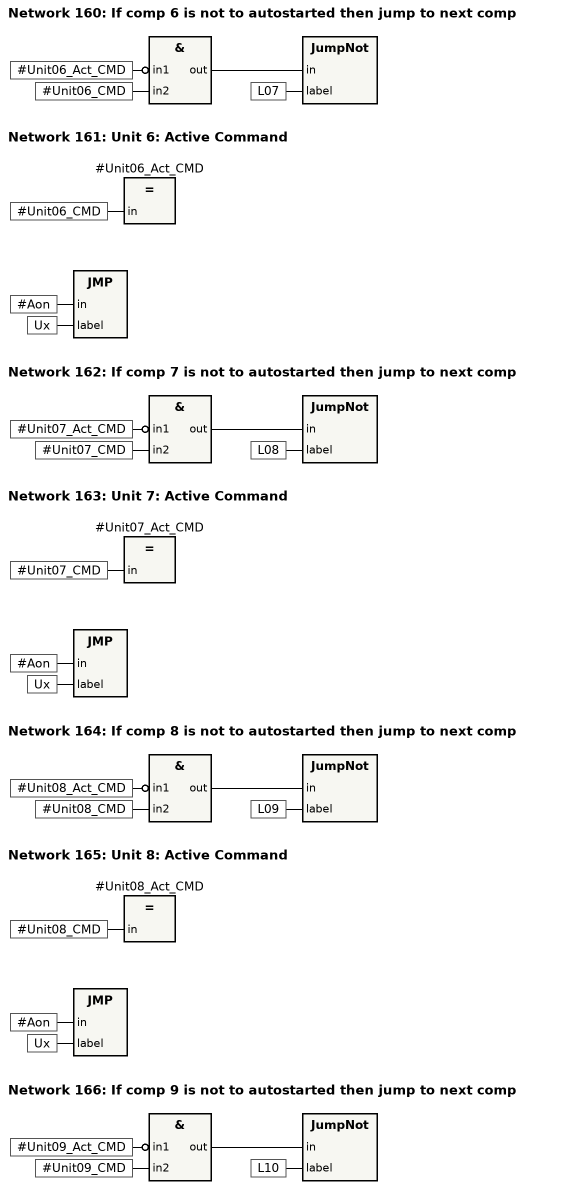
   // no SCL statement known for JumpNot: written as a call
   L06:
   JumpNot(in := NOT #Unit06_Act_CMD AND #Unit06_CMD, label := L07);
END_REGION

REGION Network 161: Unit 6: Active Command
   // Jump to end
   #Unit06_Act_CMD := #Unit06_CMD;
   IF #Aon THEN GOTO Ux; END_IF;
END_REGION

REGION Network 162: If comp 7 is not to autostarted then jump to next comp
   // no SCL statement known for JumpNot: written as a call
   L07:
   JumpNot(in := NOT #Unit07_Act_CMD AND #Unit07_CMD, label := L08);
END_REGION

REGION Network 163: Unit 7: Active Command
   // Jump to end
   #Unit07_Act_CMD := #Unit07_CMD;
   IF #Aon THEN GOTO Ux; END_IF;
END_REGION

REGION Network 164: If comp 8 is not to autostarted then jump to next comp
   // no SCL statement known for JumpNot: written as a call
   L08:
   JumpNot(in := NOT #Unit08_Act_CMD AND #Unit08_CMD, label := L09);
END_REGION

REGION Network 165: Unit 8: Active Command
   // Jump to end
   #Unit08_Act_CMD := #Unit08_CMD;
   IF #Aon THEN GOTO Ux; END_IF;
END_REGION

REGION Network 166: If comp 9 is not to autostarted then jump to next comp
   // no SCL statement known for JumpNot: written as a call
   L09:
   JumpNot(in := NOT #Unit09_Act_CMD AND #Unit09_CMD, label := L10);
END_REGION

REGION Network 167: Unit 9: Active Command
   // Jump to end
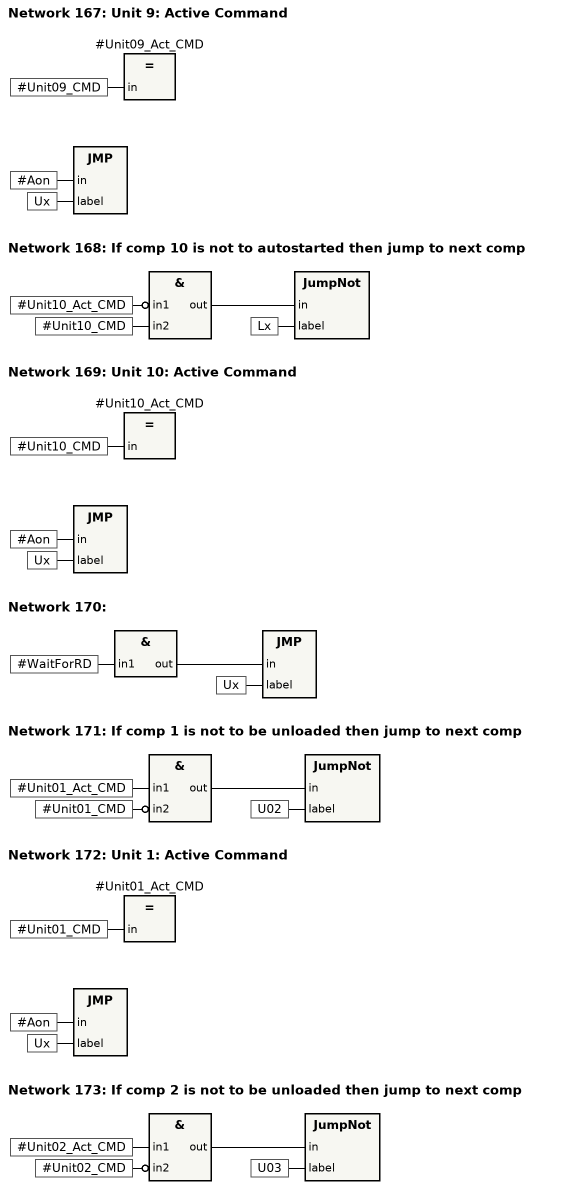
   #Unit09_Act_CMD := #Unit09_CMD;
   IF #Aon THEN GOTO Ux; END_IF;
END_REGION

REGION Network 168: If comp 10 is not to autostarted then jump to next comp
   // no SCL statement known for JumpNot: written as a call
   L10:
   JumpNot(in := NOT #Unit10_Act_CMD AND #Unit10_CMD, label := Lx);
END_REGION

REGION Network 169: Unit 10: Active Command
   // Jump to end
   #Unit10_Act_CMD := #Unit10_CMD;
   IF #Aon THEN GOTO Ux; END_IF;
END_REGION

REGION Network 170
   Lx:
   IF #WaitForRD THEN GOTO Ux; END_IF;
END_REGION

REGION Network 171: If comp 1 is not to be unloaded then jump to next comp
   // no SCL statement known for JumpNot: written as a call
   JumpNot(in := #Unit01_Act_CMD AND NOT #Unit01_CMD, label := U02);
END_REGION

REGION Network 172: Unit 1: Active Command
   #Unit01_Act_CMD := #Unit01_CMD;
   IF #Aon THEN GOTO Ux; END_IF;
END_REGION

REGION Network 173: If comp 2 is not to be unloaded then jump to next comp
   // no SCL statement known for JumpNot: written as a call
   U02:
   JumpNot(in := #Unit02_Act_CMD AND NOT #Unit02_CMD, label := U03);
END_REGION

REGION Network 174: Unit 2: Active Command
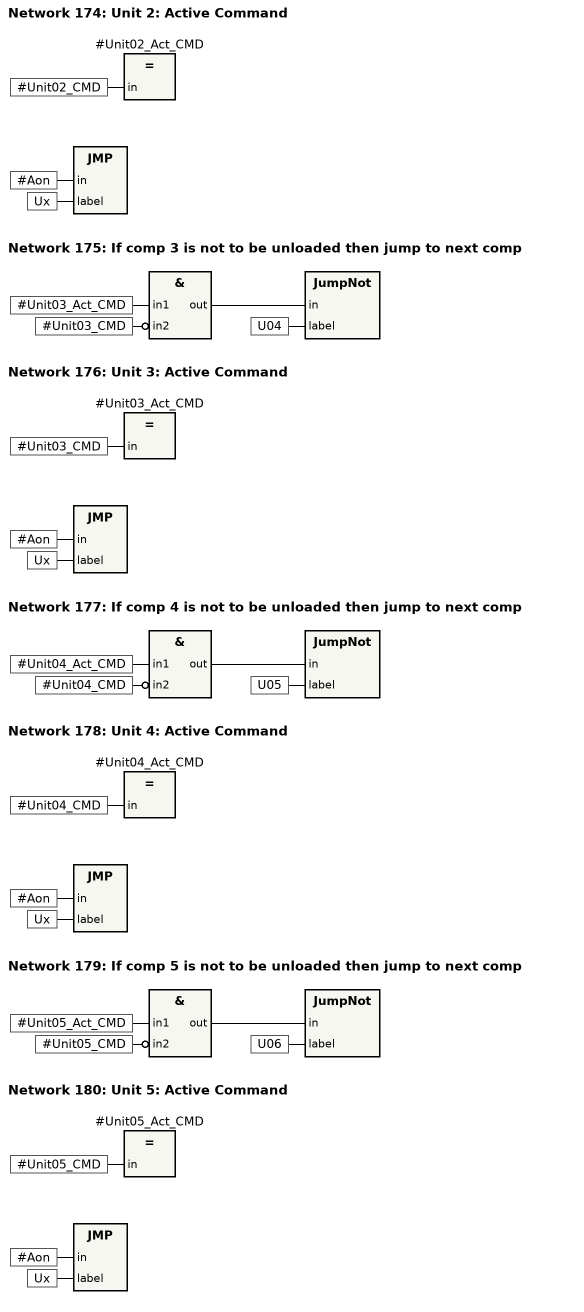
   #Unit02_Act_CMD := #Unit02_CMD;
   IF #Aon THEN GOTO Ux; END_IF;
END_REGION

REGION Network 175: If comp 3 is not to be unloaded then jump to next comp
   // no SCL statement known for JumpNot: written as a call
   U03:
   JumpNot(in := #Unit03_Act_CMD AND NOT #Unit03_CMD, label := U04);
END_REGION

REGION Network 176: Unit 3: Active Command
   #Unit03_Act_CMD := #Unit03_CMD;
   IF #Aon THEN GOTO Ux; END_IF;
END_REGION

REGION Network 177: If comp 4 is not to be unloaded then jump to next comp
   // no SCL statement known for JumpNot: written as a call
   U04:
   JumpNot(in := #Unit04_Act_CMD AND NOT #Unit04_CMD, label := U05);
END_REGION

REGION Network 178: Unit 4: Active Command
   #Unit04_Act_CMD := #Unit04_CMD;
   IF #Aon THEN GOTO Ux; END_IF;
END_REGION

REGION Network 179: If comp 5 is not to be unloaded then jump to next comp
   // no SCL statement known for JumpNot: written as a call
   U05:
   JumpNot(in := #Unit05_Act_CMD AND NOT #Unit05_CMD, label := U06);
END_REGION

REGION Network 180: Unit 5: Active Command
   #Unit05_Act_CMD := #Unit05_CMD;
   IF #Aon THEN GOTO Ux; END_IF;
END_REGION

REGION Network 181: If comp 6 is not to be unloaded then jump to next comp
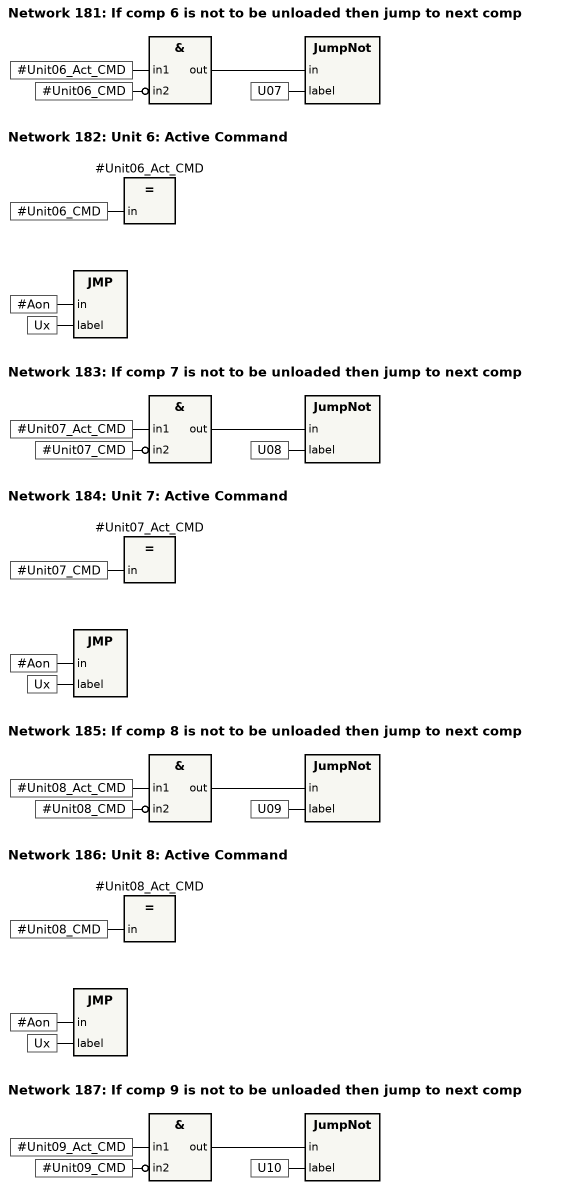
   // no SCL statement known for JumpNot: written as a call
   U06:
   JumpNot(in := #Unit06_Act_CMD AND NOT #Unit06_CMD, label := U07);
END_REGION

REGION Network 182: Unit 6: Active Command
   #Unit06_Act_CMD := #Unit06_CMD;
   IF #Aon THEN GOTO Ux; END_IF;
END_REGION

REGION Network 183: If comp 7 is not to be unloaded then jump to next comp
   // no SCL statement known for JumpNot: written as a call
   U07:
   JumpNot(in := #Unit07_Act_CMD AND NOT #Unit07_CMD, label := U08);
END_REGION

REGION Network 184: Unit 7: Active Command
   #Unit07_Act_CMD := #Unit07_CMD;
   IF #Aon THEN GOTO Ux; END_IF;
END_REGION

REGION Network 185: If comp 8 is not to be unloaded then jump to next comp
   // no SCL statement known for JumpNot: written as a call
   U08:
   JumpNot(in := #Unit08_Act_CMD AND NOT #Unit08_CMD, label := U09);
END_REGION

REGION Network 186: Unit 8: Active Command
   #Unit08_Act_CMD := #Unit08_CMD;
   IF #Aon THEN GOTO Ux; END_IF;
END_REGION

REGION Network 187: If comp 9 is not to be unloaded then jump to next comp
   // no SCL statement known for JumpNot: written as a call
   U09:
   JumpNot(in := #Unit09_Act_CMD AND NOT #Unit09_CMD, label := U10);
END_REGION

REGION Network 188: Unit 9: Active Command
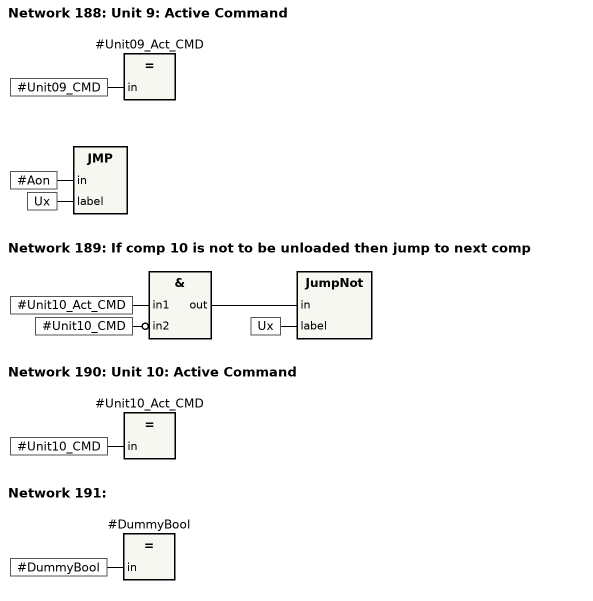
   #Unit09_Act_CMD := #Unit09_CMD;
   IF #Aon THEN GOTO Ux; END_IF;
END_REGION

REGION Network 189: If comp 10 is not to be unloaded then jump to next comp
   // no SCL statement known for JumpNot: written as a call
   U10:
   JumpNot(in := #Unit10_Act_CMD AND NOT #Unit10_CMD, label := Ux);
END_REGION

REGION Network 190: Unit 10: Active Command
   #Unit10_Act_CMD := #Unit10_CMD;
END_REGION

REGION Network 191
   Ux:
   #DummyBool := #DummyBool;
END_REGION

REGION Network 192: Reset Active commands if not selected, SACK or OK
   // Every x s a compressor is unloaded and one is loaded
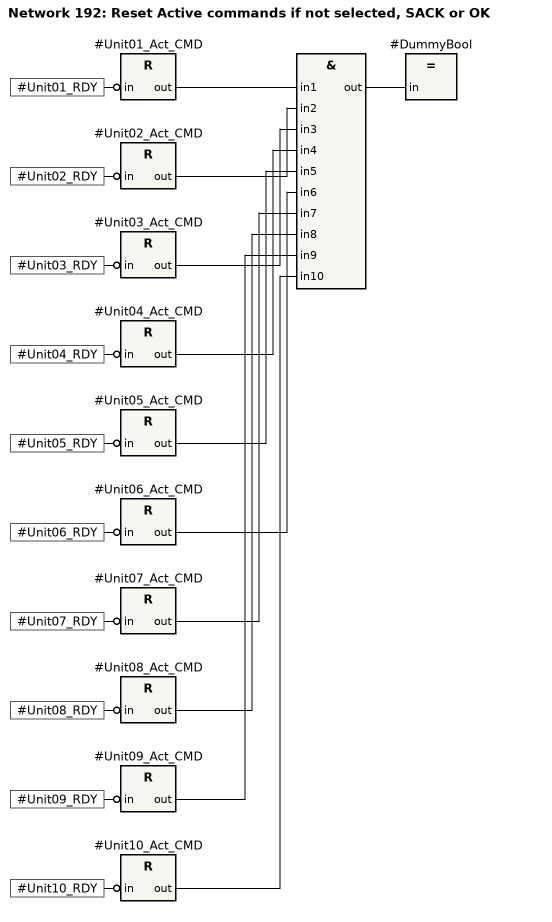
   IF NOT #Unit01_RDY THEN #Unit01_Act_CMD := FALSE; END_IF;
   IF NOT #Unit02_RDY THEN #Unit02_Act_CMD := FALSE; END_IF;
   IF NOT #Unit03_RDY THEN #Unit03_Act_CMD := FALSE; END_IF;
   IF NOT #Unit04_RDY THEN #Unit04_Act_CMD := FALSE; END_IF;
   IF NOT #Unit05_RDY THEN #Unit05_Act_CMD := FALSE; END_IF;
   IF NOT #Unit06_RDY THEN #Unit06_Act_CMD := FALSE; END_IF;
   IF NOT #Unit07_RDY THEN #Unit07_Act_CMD := FALSE; END_IF;
   IF NOT #Unit08_RDY THEN #Unit08_Act_CMD := FALSE; END_IF;
   IF NOT #Unit09_RDY THEN #Unit09_Act_CMD := FALSE; END_IF;
   IF NOT #Unit10_RDY THEN #Unit10_Act_CMD := FALSE; END_IF;
   #DummyBool := NOT #Unit01_RDY AND NOT #Unit02_RDY AND NOT #Unit03_RDY AND NOT #Unit04_RDY AND NOT #Unit05_RDY AND NOT #Unit06_RDY AND NOT #Unit07_RDY AND NOT #Unit08_RDY AND NOT #Unit09_RDY AND NOT #Unit10_RDY;
END_REGION

REGION Network 193: 12) Set Load Commands
   // Build 002 - 28 June.2019 (EXTBOB): Load outputs can only be energized if selected from faceplate
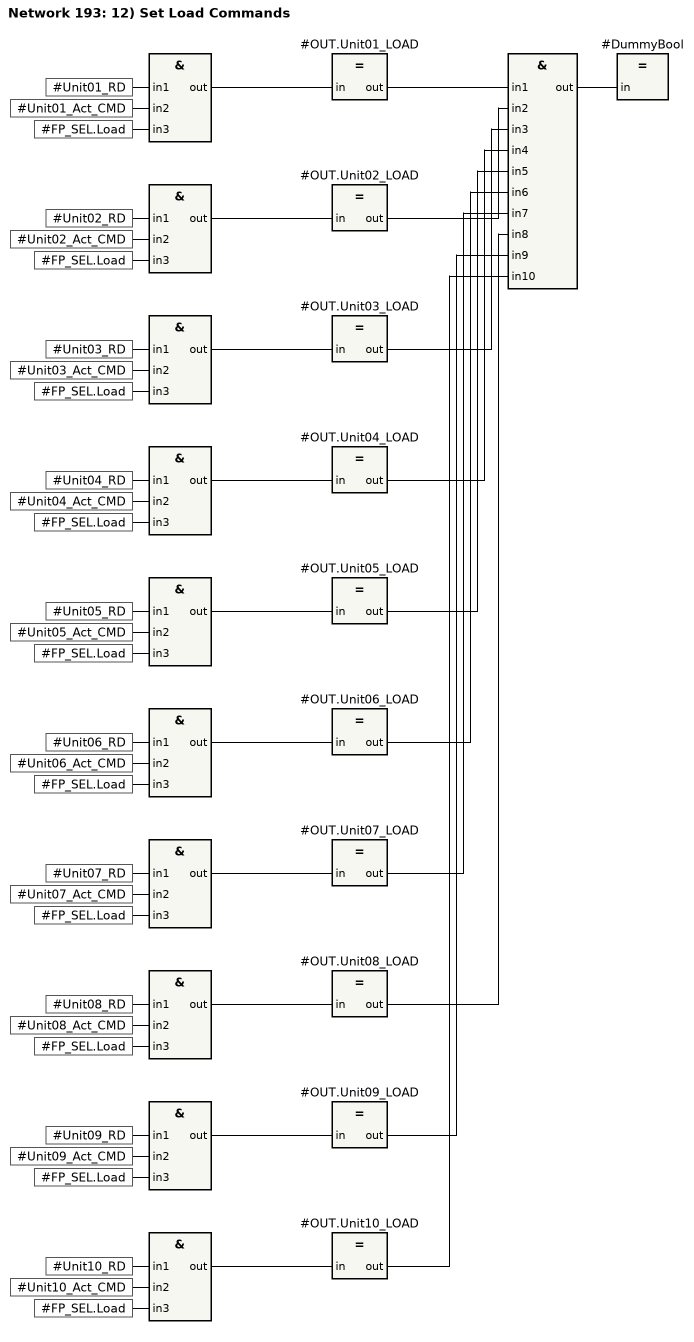
   #OUT.Unit01_LOAD := #Unit01_RD AND #Unit01_Act_CMD AND #FP_SEL.Load;
   #OUT.Unit02_LOAD := #Unit02_RD AND #Unit02_Act_CMD AND #FP_SEL.Load;
   #OUT.Unit03_LOAD := #Unit03_RD AND #Unit03_Act_CMD AND #FP_SEL.Load;
   #OUT.Unit04_LOAD := #Unit04_RD AND #Unit04_Act_CMD AND #FP_SEL.Load;
   #OUT.Unit05_LOAD := #Unit05_RD AND #Unit05_Act_CMD AND #FP_SEL.Load;
   #OUT.Unit06_LOAD := #Unit06_RD AND #Unit06_Act_CMD AND #FP_SEL.Load;
   #OUT.Unit07_LOAD := #Unit07_RD AND #Unit07_Act_CMD AND #FP_SEL.Load;
   #OUT.Unit08_LOAD := #Unit08_RD AND #Unit08_Act_CMD AND #FP_SEL.Load;
   #OUT.Unit09_LOAD := #Unit09_RD AND #Unit09_Act_CMD AND #FP_SEL.Load;
   #OUT.Unit10_LOAD := #Unit10_RD AND #Unit10_Act_CMD AND #FP_SEL.Load;
   #DummyBool := #OUT.Unit01_LOAD AND #OUT.Unit02_LOAD AND #OUT.Unit03_LOAD AND #OUT.Unit04_LOAD AND #OUT.Unit05_LOAD AND #OUT.Unit06_LOAD AND #OUT.Unit07_LOAD AND #OUT.Unit08_LOAD AND #OUT.Unit09_LOAD AND #OUT.Unit10_LOAD;
END_REGION

REGION Network 194: Set ASTR Output (Delayed off)
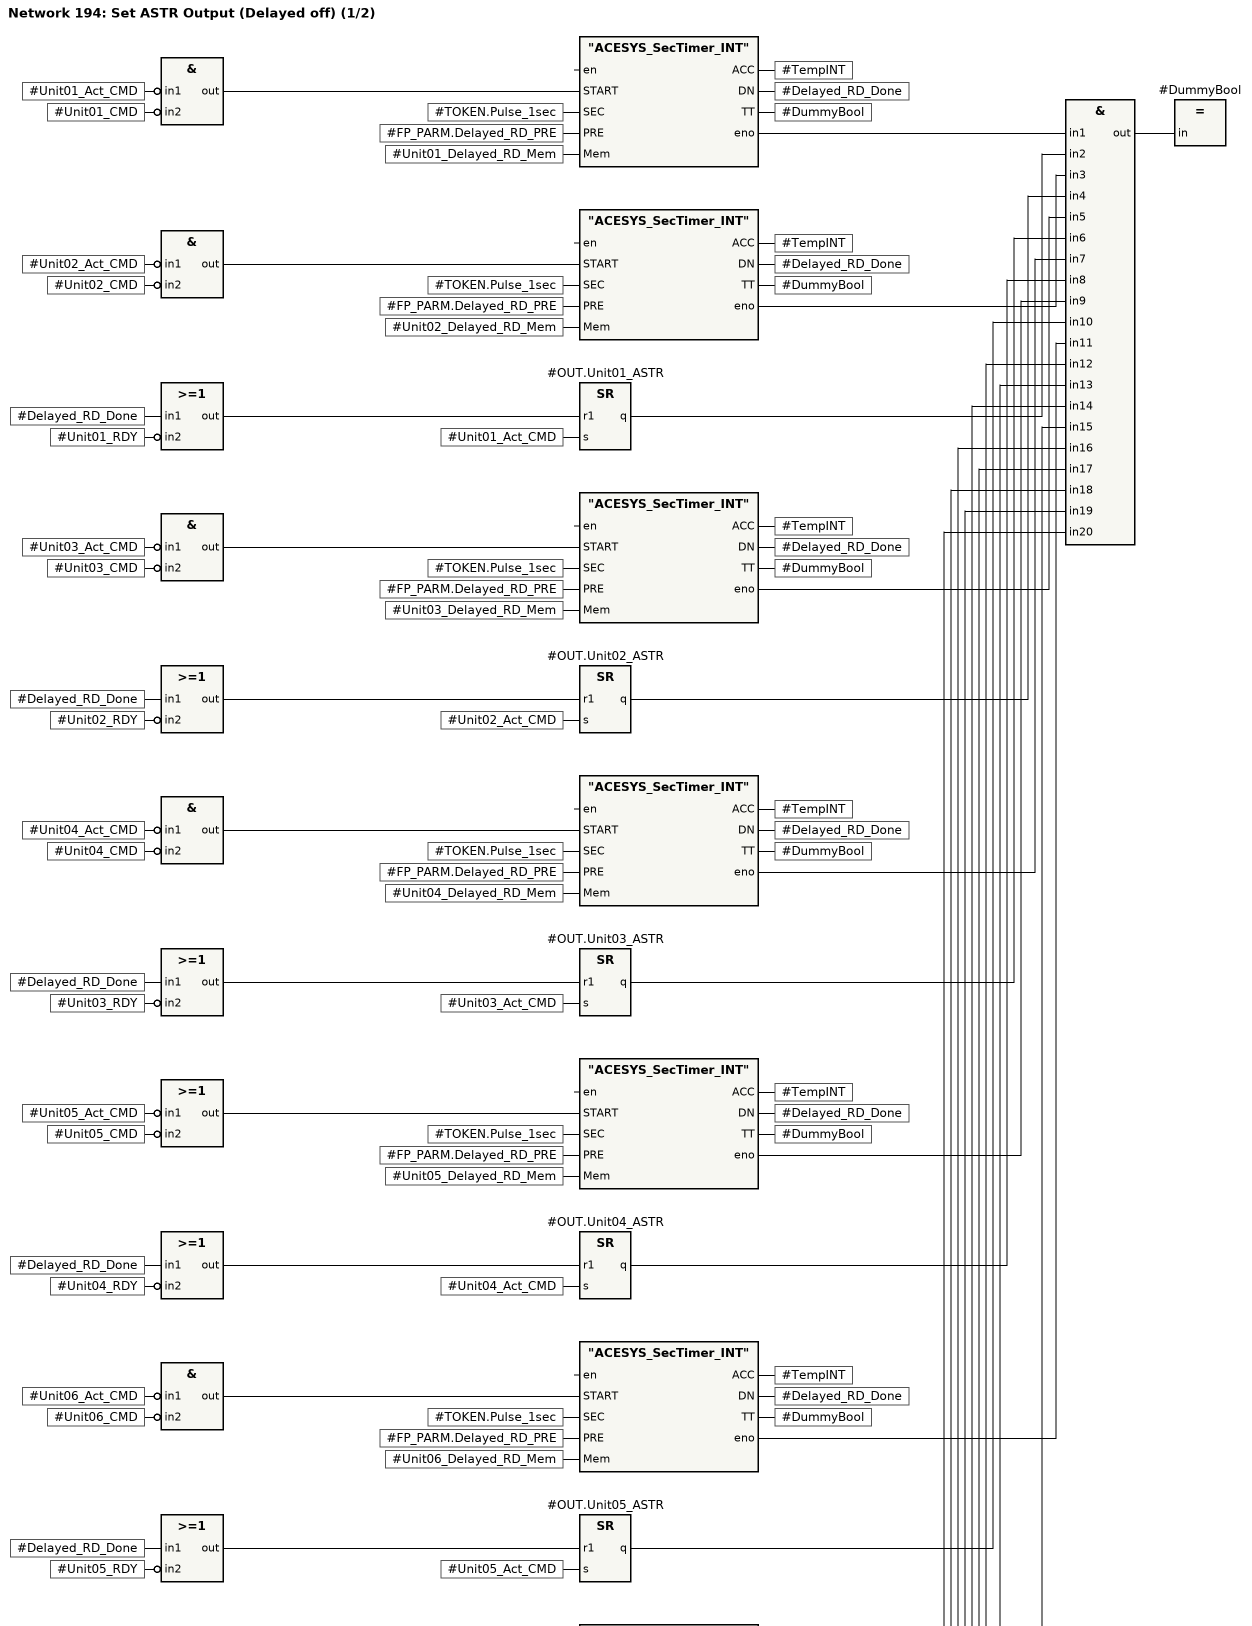
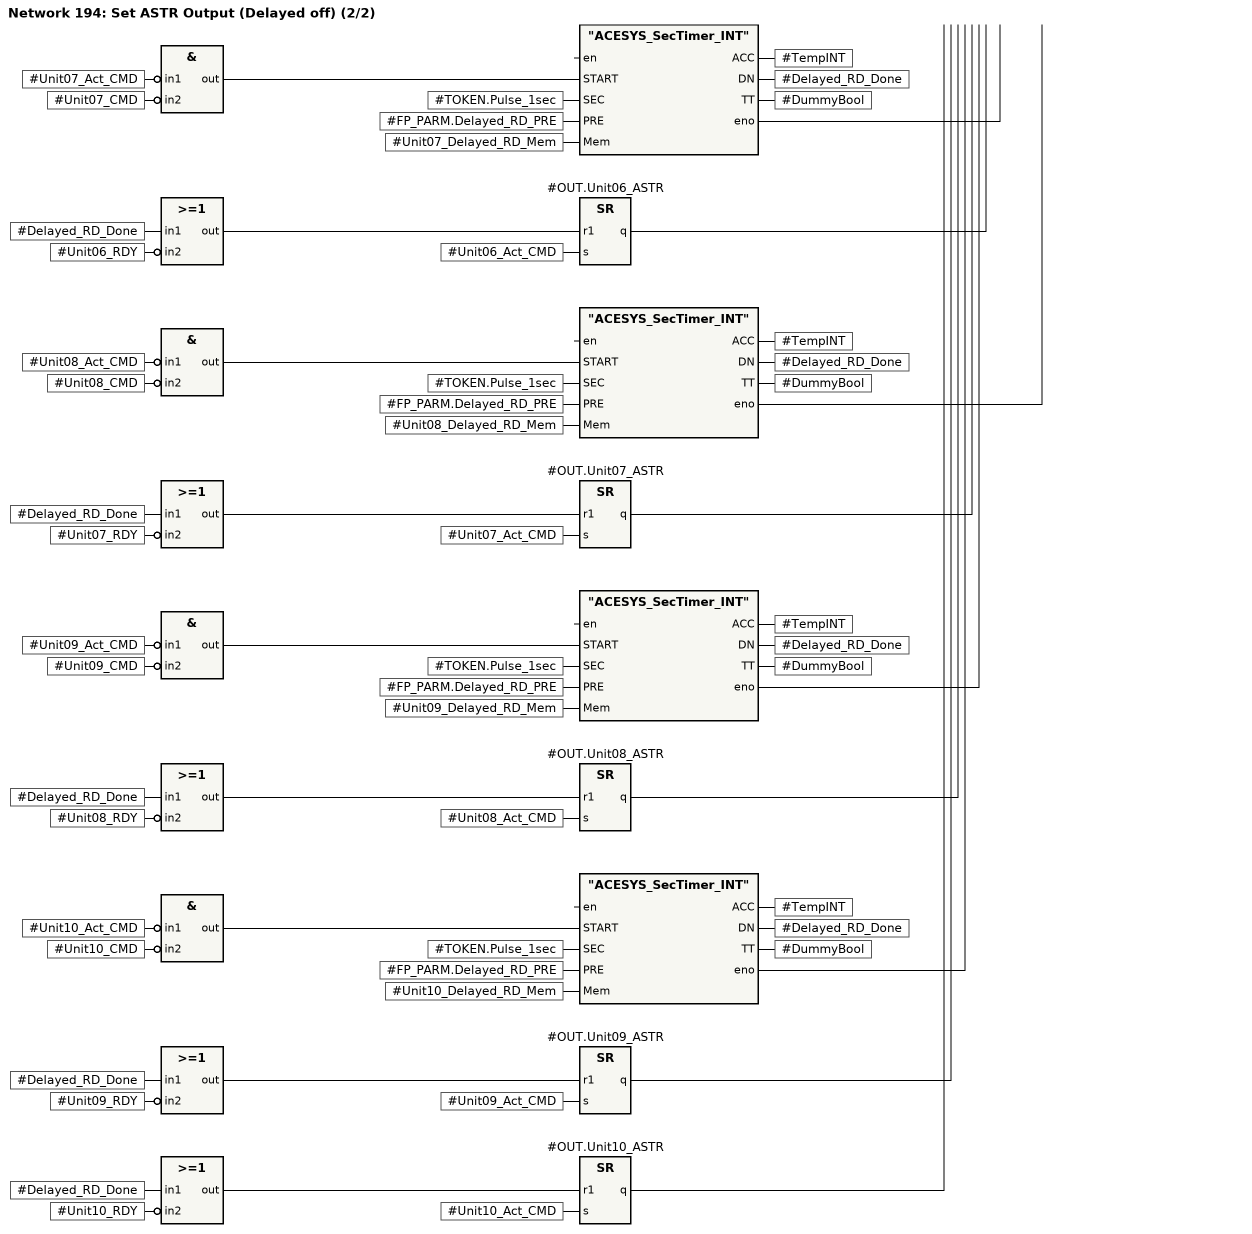
   "ACESYS_SecTimer_INT"(START := NOT #Unit01_Act_CMD AND NOT #Unit01_CMD,
                         SEC := #TOKEN.Pulse_1sec,
                         PRE := #FP_PARM.Delayed_RD_PRE,
                         Mem := #Unit01_Delayed_RD_Mem,
                         ACC => #TempINT,
                         DN => #Delayed_RD_Done,
                         TT => #DummyBool,
                         ENO => #_w1);
   IF #Unit01_Act_CMD THEN
       #OUT.Unit01_ASTR := TRUE;   // SR flip-flop
   END_IF;
   IF #Delayed_RD_Done OR NOT #Unit01_RDY THEN #OUT.Unit01_ASTR := FALSE; END_IF;
   "ACESYS_SecTimer_INT"(START := NOT #Unit02_Act_CMD AND NOT #Unit02_CMD,
                         SEC := #TOKEN.Pulse_1sec,
                         PRE := #FP_PARM.Delayed_RD_PRE,
                         Mem := #Unit02_Delayed_RD_Mem,
                         ACC => #TempINT,
                         DN => #Delayed_RD_Done,
                         TT => #DummyBool,
                         ENO => #_w2);
   IF #Unit02_Act_CMD THEN
       #OUT.Unit02_ASTR := TRUE;   // SR flip-flop
   END_IF;
   IF #Delayed_RD_Done OR NOT #Unit02_RDY THEN #OUT.Unit02_ASTR := FALSE; END_IF;
   "ACESYS_SecTimer_INT"(START := NOT #Unit03_Act_CMD AND NOT #Unit03_CMD,
                         SEC := #TOKEN.Pulse_1sec,
                         PRE := #FP_PARM.Delayed_RD_PRE,
                         Mem := #Unit03_Delayed_RD_Mem,
                         ACC => #TempINT,
                         DN => #Delayed_RD_Done,
                         TT => #DummyBool,
                         ENO => #_w3);
   IF #Unit03_Act_CMD THEN
       #OUT.Unit03_ASTR := TRUE;   // SR flip-flop
   END_IF;
   IF #Delayed_RD_Done OR NOT #Unit03_RDY THEN #OUT.Unit03_ASTR := FALSE; END_IF;
   "ACESYS_SecTimer_INT"(START := NOT #Unit04_Act_CMD AND NOT #Unit04_CMD,
                         SEC := #TOKEN.Pulse_1sec,
                         PRE := #FP_PARM.Delayed_RD_PRE,
                         Mem := #Unit04_Delayed_RD_Mem,
                         ACC => #TempINT,
                         DN => #Delayed_RD_Done,
                         TT => #DummyBool,
                         ENO => #_w4);
   IF #Unit04_Act_CMD THEN
       #OUT.Unit04_ASTR := TRUE;   // SR flip-flop
   END_IF;
   IF #Delayed_RD_Done OR NOT #Unit04_RDY THEN #OUT.Unit04_ASTR := FALSE; END_IF;
   "ACESYS_SecTimer_INT"(START := NOT #Unit05_Act_CMD OR NOT #Unit05_CMD,
                         SEC := #TOKEN.Pulse_1sec,
                         PRE := #FP_PARM.Delayed_RD_PRE,
                         Mem := #Unit05_Delayed_RD_Mem,
                         ACC => #TempINT,
                         DN => #Delayed_RD_Done,
                         TT => #DummyBool,
                         ENO => #_w5);
   IF #Unit05_Act_CMD THEN
       #OUT.Unit05_ASTR := TRUE;   // SR flip-flop
   END_IF;
   IF #Delayed_RD_Done OR NOT #Unit05_RDY THEN #OUT.Unit05_ASTR := FALSE; END_IF;
   "ACESYS_SecTimer_INT"(START := NOT #Unit06_Act_CMD AND NOT #Unit06_CMD,
                         SEC := #TOKEN.Pulse_1sec,
                         PRE := #FP_PARM.Delayed_RD_PRE,
                         Mem := #Unit06_Delayed_RD_Mem,
                         ACC => #TempINT,
                         DN => #Delayed_RD_Done,
                         TT => #DummyBool,
                         ENO => #_w6);
   IF #Unit06_Act_CMD THEN
       #OUT.Unit06_ASTR := TRUE;   // SR flip-flop
   END_IF;
   IF #Delayed_RD_Done OR NOT #Unit06_RDY THEN #OUT.Unit06_ASTR := FALSE; END_IF;
   "ACESYS_SecTimer_INT"(START := NOT #Unit07_Act_CMD AND NOT #Unit07_CMD,
                         SEC := #TOKEN.Pulse_1sec,
                         PRE := #FP_PARM.Delayed_RD_PRE,
                         Mem := #Unit07_Delayed_RD_Mem,
                         ACC => #TempINT,
                         DN => #Delayed_RD_Done,
                         TT => #DummyBool,
                         ENO => #_w7);
   IF #Unit07_Act_CMD THEN
       #OUT.Unit07_ASTR := TRUE;   // SR flip-flop
   END_IF;
   IF #Delayed_RD_Done OR NOT #Unit07_RDY THEN #OUT.Unit07_ASTR := FALSE; END_IF;
   "ACESYS_SecTimer_INT"(START := NOT #Unit08_Act_CMD AND NOT #Unit08_CMD,
                         SEC := #TOKEN.Pulse_1sec,
                         PRE := #FP_PARM.Delayed_RD_PRE,
                         Mem := #Unit08_Delayed_RD_Mem,
                         ACC => #TempINT,
                         DN => #Delayed_RD_Done,
                         TT => #DummyBool,
                         ENO => #_w8);
   IF #Unit08_Act_CMD THEN
       #OUT.Unit08_ASTR := TRUE;   // SR flip-flop
   END_IF;
   IF #Delayed_RD_Done OR NOT #Unit08_RDY THEN #OUT.Unit08_ASTR := FALSE; END_IF;
   "ACESYS_SecTimer_INT"(START := NOT #Unit09_Act_CMD AND NOT #Unit09_CMD,
                         SEC := #TOKEN.Pulse_1sec,
                         PRE := #FP_PARM.Delayed_RD_PRE,
                         Mem := #Unit09_Delayed_RD_Mem,
                         ACC => #TempINT,
                         DN => #Delayed_RD_Done,
                         TT => #DummyBool,
                         ENO => #_w9);
   IF #Unit09_Act_CMD THEN
       #OUT.Unit09_ASTR := TRUE;   // SR flip-flop
   END_IF;
   IF #Delayed_RD_Done OR NOT #Unit09_RDY THEN #OUT.Unit09_ASTR := FALSE; END_IF;
   "ACESYS_SecTimer_INT"(START := NOT #Unit10_Act_CMD AND NOT #Unit10_CMD,
                         SEC := #TOKEN.Pulse_1sec,
                         PRE := #FP_PARM.Delayed_RD_PRE,
                         Mem := #Unit10_Delayed_RD_Mem,
                         ACC => #TempINT,
                         DN => #Delayed_RD_Done,
                         TT => #DummyBool,
                         ENO => #_w10);
   IF #Unit10_Act_CMD THEN
       #OUT.Unit10_ASTR := TRUE;   // SR flip-flop
   END_IF;
   IF #Delayed_RD_Done OR NOT #Unit10_RDY THEN #OUT.Unit10_ASTR := FALSE; END_IF;
   #DummyBool := #_w1 AND #OUT.Unit01_ASTR AND #_w2 AND #OUT.Unit02_ASTR AND #_w3 AND #OUT.Unit03_ASTR AND #_w4 AND #OUT.Unit04_ASTR AND #_w5 AND #OUT.Unit05_ASTR AND #_w6 AND #OUT.Unit06_ASTR AND #_w7 AND #OUT.Unit07_ASTR AND #_w8 AND #OUT.Unit08_ASTR AND #_w9 AND #OUT.Unit09_ASTR AND #_w10 AND #OUT.Unit10_ASTR;
END_REGION

REGION Network 195
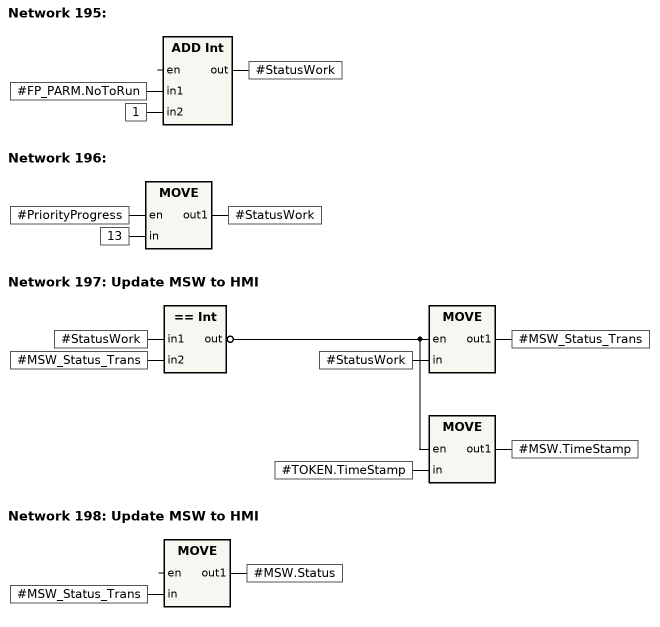
   #StatusWork := #FP_PARM.NoToRun + 1;
END_REGION

REGION Network 196
   IF #PriorityProgress THEN #StatusWork := 13; END_IF;
END_REGION

REGION Network 197: Update MSW to HMI
   #_w1 := NOT (#StatusWork = #MSW_Status_Trans);
   IF #_w1 THEN
       #MSW_Status_Trans := #StatusWork;
       #MSW.TimeStamp := #TOKEN.TimeStamp;
   END_IF;
END_REGION

REGION Network 198: Update MSW to HMI
   #MSW.Status := #MSW_Status_Trans;
END_REGION

REGION Network 199: Write STAT to OUT
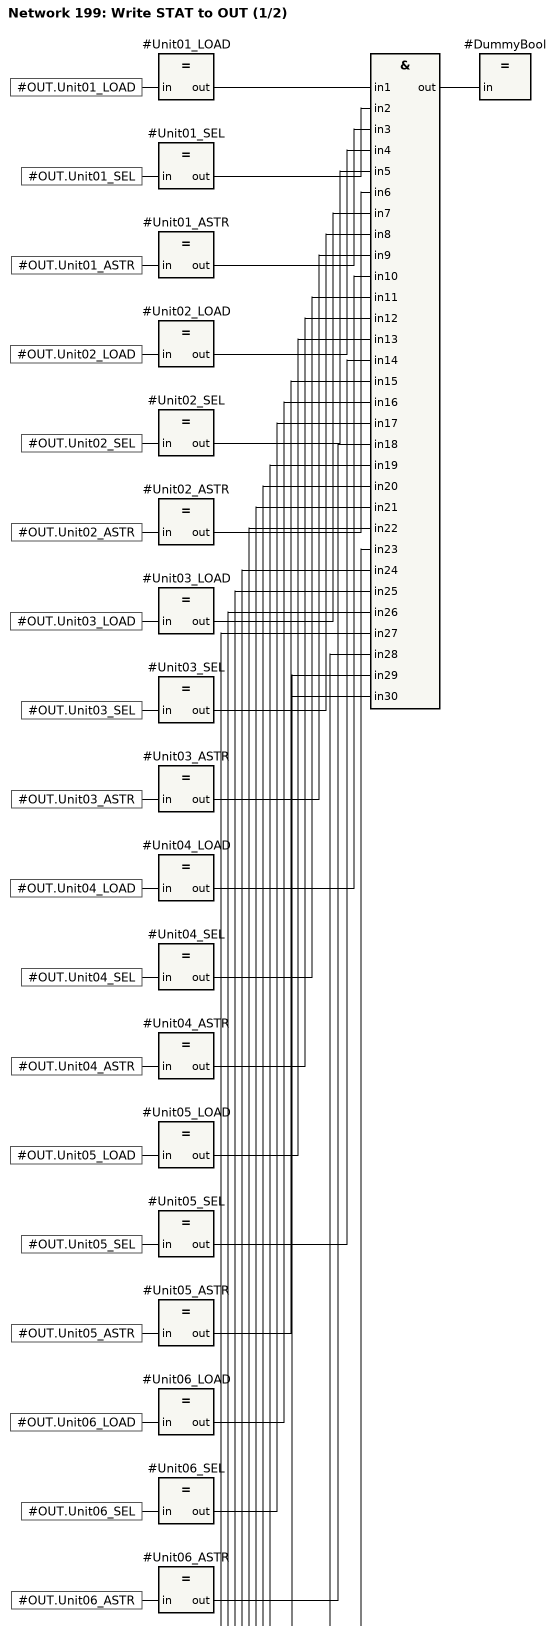
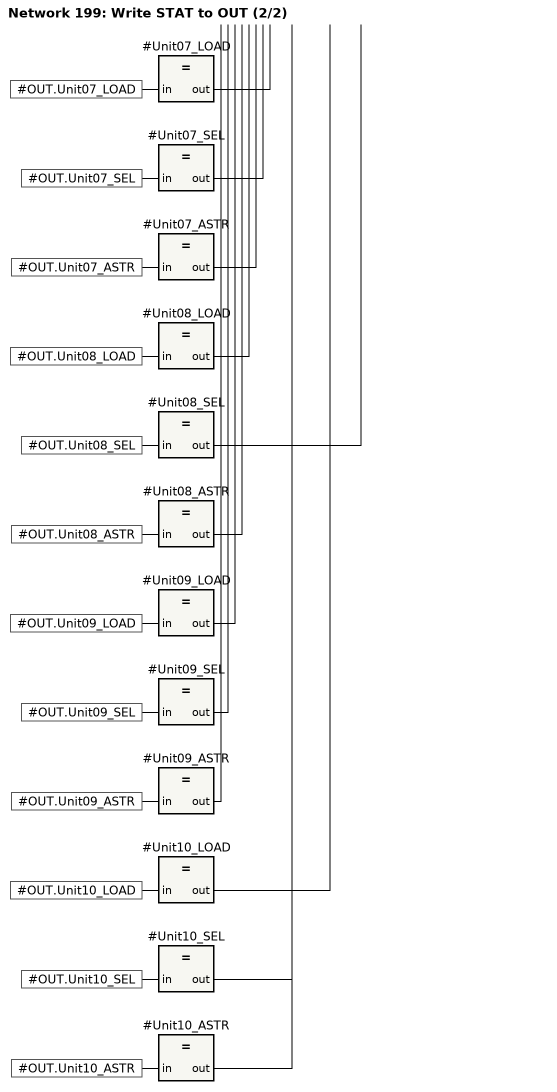
   #Unit01_LOAD := #OUT.Unit01_LOAD;
   #Unit01_SEL := #OUT.Unit01_SEL;
   #Unit01_ASTR := #OUT.Unit01_ASTR;
   #Unit02_LOAD := #OUT.Unit02_LOAD;
   #Unit02_SEL := #OUT.Unit02_SEL;
   #Unit02_ASTR := #OUT.Unit02_ASTR;
   #Unit03_LOAD := #OUT.Unit03_LOAD;
   #Unit03_SEL := #OUT.Unit03_SEL;
   #Unit03_ASTR := #OUT.Unit03_ASTR;
   #Unit04_LOAD := #OUT.Unit04_LOAD;
   #Unit04_SEL := #OUT.Unit04_SEL;
   #Unit04_ASTR := #OUT.Unit04_ASTR;
   #Unit05_LOAD := #OUT.Unit05_LOAD;
   #Unit05_SEL := #OUT.Unit05_SEL;
   #Unit05_ASTR := #OUT.Unit05_ASTR;
   #Unit06_LOAD := #OUT.Unit06_LOAD;
   #Unit06_SEL := #OUT.Unit06_SEL;
   #Unit06_ASTR := #OUT.Unit06_ASTR;
   #Unit07_LOAD := #OUT.Unit07_LOAD;
   #Unit07_SEL := #OUT.Unit07_SEL;
   #Unit07_ASTR := #OUT.Unit07_ASTR;
   #Unit08_LOAD := #OUT.Unit08_LOAD;
   #Unit08_SEL := #OUT.Unit08_SEL;
   #Unit08_ASTR := #OUT.Unit08_ASTR;
   #Unit09_LOAD := #OUT.Unit09_LOAD;
   #Unit09_SEL := #OUT.Unit09_SEL;
   #Unit09_ASTR := #OUT.Unit09_ASTR;
   #Unit10_LOAD := #OUT.Unit10_LOAD;
   #Unit10_SEL := #OUT.Unit10_SEL;
   #Unit10_ASTR := #OUT.Unit10_ASTR;
   #DummyBool := #OUT.Unit01_LOAD AND #OUT.Unit01_SEL AND #OUT.Unit01_ASTR AND #OUT.Unit02_LOAD AND #OUT.Unit02_SEL AND #OUT.Unit02_ASTR AND #OUT.Unit03_LOAD AND #OUT.Unit03_SEL AND #OUT.Unit03_ASTR AND #OUT.Unit04_LOAD AND #OUT.Unit04_SEL AND #OUT.Unit04_ASTR AND #OUT.Unit05_LOAD AND #OUT.Unit05_SEL AND #OUT.Unit05_ASTR AND #OUT.Unit06_LOAD AND #OUT.Unit06_SEL AND #OUT.Unit06_ASTR AND #OUT.Unit07_LOAD AND #OUT.Unit07_SEL AND #OUT.Unit07_ASTR AND #OUT.Unit08_LOAD AND #OUT.Unit08_SEL AND #OUT.Unit08_ASTR AND #OUT.Unit09_LOAD AND #OUT.Unit09_SEL AND #OUT.Unit09_ASTR AND #OUT.Unit10_LOAD AND #OUT.Unit10_SEL AND #OUT.Unit10_ASTR;
END_REGION
END_FUNCTION_BLOCK

FUNCTION_BLOCK "ACESYS_PIACS"   // FB233, FBD
TITLE = ACESYS V8.0 - Build 001 - PIACS
{ S7_Optimized_Access := 'FALSE' }
AUTHOR : FLSmidth
FAMILY : ACESYS
NAME : PIACS
VERSION : 8.0
   VAR_INPUT
      INREF : Int;   // Input address
      OUTREF : Int;   // Output address
      NET : Int;   // Fieldbus Network Ref.
      NODE : Int;   // Fieldbus Node Ref.
      FuncType : Int;   // Function Type (1=Type1; 2=Type2;.....)
      Options : Int;   // Function Options (1=Option1; 2=Option2......)
      ARM : Bool;   // ARM active
      COmax2 : Bool;   // COmax2 interlock (0=Interlocked)
      KAPulseLength : Int;   // Keep alive pulse length
   END_VAR
   VAR_OUTPUT
      UDC_Sec : Real;   // UDC Rectifier voltage Section(0-100%)
      IDC_Sec : Real;   // IDC Rectifier current Section(0-100%)
      MSW : "ACESYS_HMI_STAT_32T";
   END_VAR
   VAR_IN_OUT
      TOKEN : "ACESYS_TOKEN";
   END_VAR
   VAR
      BlockInfo : Struct
         Ace_Version : Int;   // Acesys Block Version Number
         Ace_BuildNo : Int;   // Acesys Block Build Number
         DB_Number : Int;   // Block Instance DB Number
         PIACS_Version : Int;
      END_STRUCT;
      FP_CMD : Struct   // Faceplate Commands
         Spare_08 : Bool;
         Spare_09 : Bool;
         Spare_10 : Bool;
         Spare_11 : Bool;
         Spare_12 : Bool;
         Spare_13 : Bool;
         Spare_14 : Bool;
         AckAlarm : Bool;   // Alarm Acknowledge
         Spare_00 : Bool;
         Spare_01 : Bool;
         Spare_02 : Bool;
         Spare_03 : Bool;
         Spare_04 : Bool;
         Spare_05 : Bool;
         Spare_06 : Bool;
         Spare_07 : Bool;
      END_STRUCT;
      SectionIn : Struct
         I000_0 : Bool;
         I000_1 : Bool;
         I000_2 : Bool;
         I000_3 : Bool;
         I000_4 : Bool;
         I000_5 : Bool;
         I000_6 : Bool;
         I000_7 : Bool;
         I001_0 : Bool;   // PIACS Life OK "1"
         I001_1 : Bool;   // Gateway OK "1"
         I001_2 : Bool;
         I001_3 : Bool;
         I001_4 : Bool;
         I001_5 : Bool;
         I001_6 : Bool;
         I001_7 : Bool;
         IW002 : Int;   // PIACS Software version
         IW004 : Int;   // Life Signal Pulse Time
         IW006 : Int;
         IW008 : Int;
         I010_0 : Bool;
         I010_1 : Bool;
         I010_2 : Bool;   // TR COmax2 active "1"
         I010_3 : Bool;
         I010_4 : Bool;
         I010_5 : Bool;
         I010_6 : Bool;
         I010_7 : Bool;
         I011_0 : Bool;   // TR Warning "1"
         I011_1 : Bool;   // TR ready "1"
         I011_2 : Bool;   // TR on "1"
         I011_3 : Bool;   // TR COmax3 active "1"
         I011_4 : Bool;   // TR reset ACKnowledge "1"
         I011_5 : Bool;
         I011_6 : Bool;
         I011_7 : Bool;   // ARM active "1"
         I012_0 : Bool;   // TR undervoltage 30s "1"
         I012_1 : Bool;   // TR overvoltage 1s "1"
         I012_2 : Bool;   // TR µP check error "1"
         I012_3 : Bool;   // TR mains sync.failure "1"
         I012_4 : Bool;   // TR low temperature E1 / E2 "1"
         I012_5 : Bool;
         I012_6 : Bool;
         I012_7 : Bool;
         I013_0 : Bool;   // TR interlocking "1"
         I013_1 : Bool;   // TR high pressure oil tank "1"
         I013_2 : Bool;   // TR high temoerature oil tank "1"
         I013_3 : Bool;   // TR low oil level "1"
         I013_4 : Bool;   // TR set grounded "1"
         I013_5 : Bool;   // TR optional alarm "1"
         I013_6 : Bool;   // TR mains overload "1"
         I013_7 : Bool;   // TR start failure "1"
         I014_0 : Bool;   // Rapping timer 1 failure "1"
         I014_1 : Bool;
         I014_2 : Bool;   // Rapping timer 2 on "1"
         I014_3 : Bool;   // Rapping timer 2 failure "1"
         I014_4 : Bool;
         I014_5 : Bool;   // Rapping timer 3 on "1"
         I014_6 : Bool;
         I014_7 : Bool;   // Rapping timer 3 failure "1"
         I015_0 : Bool;   // Rapping Warning "1"
         I015_1 : Bool;   // Rapping ready "1"
         I015_2 : Bool;   // Rapping on "1"
         I015_3 : Bool;   // Rapping local command "1"
         I015_4 : Bool;   // Rapping reset ACKnowledge "1"
         I015_5 : Bool;
         I015_6 : Bool;
         I015_7 : Bool;   // Rapping timer 1 on "1"
         I016_0 : Bool;
         I016_1 : Bool;   // T1 Interlock
         I016_2 : Bool;
         I016_3 : Bool;   // T2 Interlock
         I016_4 : Bool;
         I016_5 : Bool;   // T3 Interlock
         I016_6 : Bool;
         I016_7 : Bool;
         I017_0 : Bool;   // Rapping group interlock "1"
         I017_1 : Bool;   // Rapping feedback failure T1
         I017_2 : Bool;   // Rapping mains failure T1
         I017_3 : Bool;   // Rapping feedback failure T2
         I017_4 : Bool;   // Rapping mains failure T2
         I017_5 : Bool;   // Rapping feedback failure T3
         I017_6 : Bool;   // Rapping mains failure T3
         I017_7 : Bool;   // Rapping start failure "1"
         I018_0 : Bool;   // Heating E1 failure "1"
         I018_1 : Bool;
         I018_2 : Bool;   // Heating E2 on "1"
         I018_3 : Bool;   // Heating E2 failure "1"
         I018_4 : Bool;
         I018_5 : Bool;   // Heating E3 on "1"
         I018_6 : Bool;
         I018_7 : Bool;   // Heating E3 failure "1"
         I019_0 : Bool;   // Heating Warning "1"
         I019_1 : Bool;   // Heating Ready "1"
         I019_2 : Bool;   // Heating On "1"
         I019_3 : Bool;   // Heating local command "1"
         I019_4 : Bool;   // Heating reset ACKnowledge "1"
         I019_5 : Bool;
         I019_6 : Bool;
         I019_7 : Bool;   // Heating E1 on "1"
         I020_0 : Bool;
         I020_1 : Bool;   // Heating E1 sens. Failure "1"
         I020_2 : Bool;   // Heating E1 low temperature warning "1"
         I020_3 : Bool;   // Heating E2 sens. Failure "1"
         I020_4 : Bool;   // Heating E2 low temperature warning "1"
         I020_5 : Bool;   // Heating E3 sens. Failure "1"
         I020_6 : Bool;
         I020_7 : Bool;   // Heating E3 low temperature warning "1"
         I021_0 : Bool;   // Heating Group interlock "1"
         I021_1 : Bool;   // Heating Feedback failure E1 "1"
         I021_2 : Bool;   // Heating Overload E1 "1"
         I021_3 : Bool;   // Heating Feedback failure E2 "1"
         I021_4 : Bool;   // Heating Overload failure E2 "1"
         I021_5 : Bool;   // Heating Feedback failure E3 "1"
         I021_6 : Bool;   // Heating Overload failure E3 "1"
         I021_7 : Bool;   // Heating Start failure "1"
         IW022 : Int;
         IW024 : Int;
         IW026 : Int;
         IW028 : Int;   // NEC 1,3,5..25
         IW030 : Int;   // Rectifier voltage Udc 0-7440a) = 0-xxx kV)
         IW032 : Int;   // Rectifier min. voltage Udc 0-7440a) ( 0-xxx kV )
         IW034 : Int;
         IW036 : Int;   // Rectifier secondary current Idc 0-7440a) = 0-xxx mA
         IW038 : Int;   // Rect. primary current Iprim 0-4000b) = 0-xxx Arms
         IW040 : Int;
         IW042 : Int;   // Rectifier sparkrate 0-9999 ( 0 - 999.9 /min )
         IW044 : Int;
         IW046 : Int;
         IW048 : Int;
         IW050 : Int;
         IW052 : Int;
         IW054 : Int;
         IW056 : Int;   // Rectifier Idc_Limit 0-3000 mA
         IW058 : Int;   // Rectifier ARM_I_limit 0-3000 mA
         IW060 : Int;
         IW062 : Int;
         IW064 : Int;
         IW066 : Int;
         IW068 : Int;
         IW070 : Int;
         IW072 : Int;
         IW074 : Int;
         IW076 : Int;
         IW078 : Int;
         IW080 : Int;
         IW082 : Int;
         IW084 : Int;
         IW086 : Int;
         IW088 : Int;
         IW090 : Int;
         IW092 : Int;
         IW094 : Int;
         IW096 : Int;   // Rectifier Optim_Mode 00..21 ( ILim#, Nec# )
         IW098 : Int;   // Rectifier ARM_Optim_Mode 00..21 ( ILim#, Nec# )
      END_STRUCT;
      SectionOut : Struct
         Q000_0 : Bool;
         Q000_1 : Bool;
         Q000_2 : Bool;
         Q000_3 : Bool;
         Q000_4 : Bool;
         Q000_5 : Bool;
         Q000_6 : Bool;
         Q000_7 : Bool;
         Q001_0 : Bool;   // Handshake "1","0"..."1" to ESP system
         Q001_1 : Bool;
         Q001_2 : Bool;
         Q001_3 : Bool;
         Q001_4 : Bool;
         Q001_5 : Bool;
         Q001_6 : Bool;
         Q001_7 : Bool;
         QW002 : Int;
         Q004_0 : Bool;
         Q004_1 : Bool;   // CO_max2_Cmd
         Q004_2 : Bool;
         Q004_3 : Bool;
         Q004_4 : Bool;
         Q004_5 : Bool;
         Q004_6 : Bool;
         Q004_7 : Bool;
         Q005_0 : Bool;
         Q005_1 : Bool;
         Q005_2 : Bool;
         Q005_3 : Bool;   // TR command "1" (COMax3)
         Q005_4 : Bool;   // TR reset "1"
         Q005_5 : Bool;
         Q005_6 : Bool;   // ARM_Cmd
         Q005_7 : Bool;
         Q006_0 : Bool;
         Q006_1 : Bool;
         Q006_2 : Bool;
         Q006_3 : Bool;
         Q006_4 : Bool;
         Q006_5 : Bool;
         Q006_6 : Bool;
         Q006_7 : Bool;
         Q007_0 : Bool;
         Q007_1 : Bool;
         Q007_2 : Bool;
         Q007_3 : Bool;   // Rapping command "1"
         Q007_4 : Bool;   // Rapping reset "1"
         Q007_5 : Bool;
         Q007_6 : Bool;
         Q007_7 : Bool;
         Q008_0 : Bool;
         Q008_1 : Bool;
         Q008_2 : Bool;
         Q008_3 : Bool;
         Q008_4 : Bool;
         Q008_5 : Bool;
         Q008_6 : Bool;
         Q008_7 : Bool;
         Q009_0 : Bool;
         Q009_1 : Bool;
         Q009_2 : Bool;
         Q009_3 : Bool;   // Heating command "1"
         Q009_4 : Bool;   // Heating reset
         Q009_5 : Bool;
         Q009_6 : Bool;
         Q009_7 : Bool;
         QW010 : Int;
         QW012 : Int;
         QW014 : Int;
         QW016 : Int;
         QW018 : Int;   // Rectifier Idc_Limit 0-3000 mA
         QW020 : Int;   // Rectifier ARM_I_limit 0-3000 mA
         QW022 : Int;
         QW024 : Int;
         QW026 : Int;
         QW028 : Int;
         QW030 : Int;
         QW032 : Int;
         QW034 : Int;
         QW036 : Int;
         QW038 : Int;
         QW040 : Int;
         QW042 : Int;
         QW044 : Int;
         QW046 : Int;
         QW048 : Int;
         QW050 : Int;
         QW052 : Int;
         QW054 : Int;
         QW056 : Int;
         QW058 : Int;   // Rectifier Optim_Mode 00..21 ( ILim#, Nec# )
         QW060 : Int;   // Rectifier ARM_Optim_Mode 00..21 ( ILim#, Nec# )
      END_STRUCT;
      ECSscaledValues : Struct
         ECS_UDCSec : Int;   // Scaled UDC to ECS
         ECS_UDCMinSec : Int;   // Scaled UDC min to ECS
         ECS_IDCSec : Int;   // Scaled IDC to ECS
         ECS_IprimSec : Int;   // Scaled IDC to ECS
      END_STRUCT;
      ScaleValues : Struct
         Select50Hz : Bool;   // Frequency selected
         Select60Hz : Bool;   // Frequency selected
         UDCScaleSec : Real;   // UDC Scale value
         IDCScaleSec : Real;   // IDC Scale value
         IPrimScaleSec : Real;   // IPrim Scale value
      END_STRUCT;
      FP_SIM : "ACESYS_SIM_PIACS";
      ONS : Struct
         KA_Pulse : Bool;
         Hz50 : Bool;
         Hz60 : Bool;
         AckAlarm : Bool;
      END_STRUCT;
      AlarmNo : Int;
      AlarmNo_Old : Int;
      StatusWork : Int;
      KAPulseTimer : Int;   // Keep alive pulsetimer
      KAPulse : Bool;   // Keep alive pulse
      AckTRSec : Bool;   // Latched acknowledeg TR
      AckRapSec : Bool;   // Latched acknowledeg rapping
      AckHeatSec : Bool;   // Latched acknowledeg heating
      ALARM_AlarmPresent : Bool;
      ALARM_WarnPresent : Bool;
      ALARM_FailureAckRequired : Bool;
      ALARM_WarnAckRequired : Bool;
      CMD_AckAlarm : Bool;
      MSW_EXT_AlarmFailUnAck : Bool;
      MSW_Status_Trans : Int;
   END_VAR
   VAR_TEMP
      BLOCK_RET_VAL : Int;
      ScaleConstantSec : Real;   // Scale constant UDC and IDC
      ScaleConstantPrim : Real;   // Scale constant Iprim
      TempReal : Real;
      Aon : Bool;
      Aoff : Bool;
      DummyBool : Bool;
      KAPulseHelp : Bool;   // Keep alive pulse help bit
      DB_Pointer : ANY;
      IO_Pointer : ANY;
      Addr_InstanceDB : DWord;
      TempDword : DWord;
      TempReal_1 : Real;
   END_VAR
   VAR_TEMP   // added for the SCL form of the ladder/FBD networks
      _w1 : Bool;
      _w2 : Bool;
   END_VAR
BEGIN

REGION Network 1
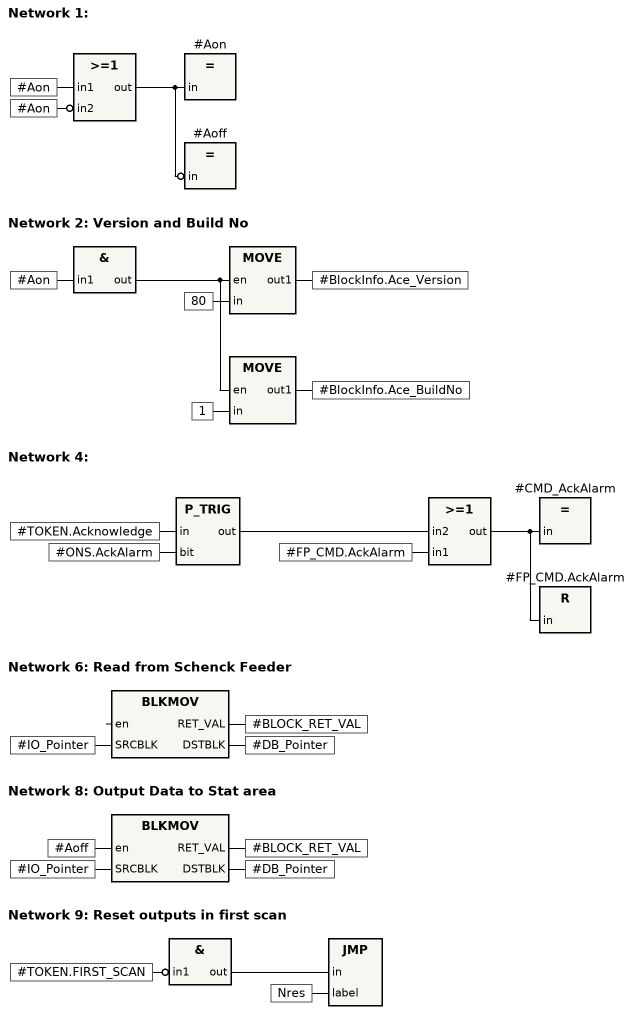
   #Aon := #Aon OR NOT #Aon;
   #Aoff := NOT #Aon;
END_REGION

REGION Network 2: Version and Build No
   IF #Aon THEN
       #BlockInfo.Ace_Version := 80;
       #BlockInfo.Ace_BuildNo := 1;
   END_IF;
END_REGION

REGION Network 3 (STL): Instance DB Number to Faceplate
         L     DINO;
         T     #BlockInfo.DB_Number;
END_REGION

REGION Network 4
   #_w1 := #TOKEN.Acknowledge AND NOT #ONS.AckAlarm;   // rising edge
   #ONS.AckAlarm := #TOKEN.Acknowledge;
   #CMD_AckAlarm := #_w1 OR #FP_CMD.AckAlarm;
   IF #CMD_AckAlarm THEN #FP_CMD.AckAlarm := FALSE; END_IF;
END_REGION

REGION Network 5 (STL): Target Pointers Recieve input data
         LAR1;  // Make AR1 point to calling program stack
         L     16#10;  // ANY Syntax ID
         T     LB[AR1, P#0.0];  // ..Store Byte 0
         L     16#02;  // Data Type = Byte
         T     LB[AR1, P#1.0];  // ..Store Byte 1
         L     100;  // Load Packed length
         T     LW[AR1, P#2.0];  // ..Store byte 2/3
         L     0;  // used with DB else "0"
         T     LW[AR1, P#4.0];  // ..Store byte 4/5
         L     #INREF;  // Source offset (Variable for Node's)
         SLD   3;  // with offset
         OD    16#8100_0000;  // Input Area (I/O) Code (S7)
         T     LD[AR1, P#6.0];  // ..Store byte 6/7/8/9

         LAR1;  // Load start point of cyclic data
         TAR1  #TempDword;  // Store in temp. point
         L     #TempDword;  // Load temp. point
         T     #Addr_InstanceDB;  // Store start point as DB address

         LAR1;  // Make AR1 point to calling program stack
         L     16#10;  // ANY Syntax ID
         T     LB[AR1, P#0.0];  // ..Store Byte 0
         L     16#02;  // Data Type = Byte
         T     LB[AR1, P#1.0];  // ..Store Byte 1
         L     100;  // Load Packed length
         T     LW[AR1, P#2.0];  // ..Store Byte 2/3
         L     #BlockInfo.DB_Number;  // used with DB use No. else "0"
         T     LW[AR1, P#4.0];  // ..Store byte 4/5
         L     #Addr_InstanceDB;  // Load Instance DB Start address
         L     16#8500_0000;
         -D;
         L     16#8400_0000;
         +D;
         T     LD[AR1, P#6.0];  // ..Store byte 6/7/8/9
END_REGION

REGION Network 6: Read from Schenck Feeder
   #BLOCK_RET_VAL := BLKMOV(SRCBLK := #IO_Pointer, DSTBLK => #DB_Pointer);
END_REGION

REGION Network 7 (STL): Target Pointers Sending Output Data
         LAR1;  // Make AR1 pointer to Unit Output
         L     16#10;  // ANY Syntax ID
         T     LB[AR1, P#0.0];  // ..Store Byte 0
         L     16#02;  // Data Type = Byte
         T     LB[AR1, P#1.0];  // ..Store Byte 1
         L     62;  // Load Packed length
         T     LW[AR1, P#2.0];  // ..Store byte 2/3
         L     0;  // used with DB else "0"
         T     LW[AR1, P#4.0];  // ..Store byte 4/5
         L     #OUTREF;  // Source offset (Variable for Node's)
         SLD   3;  // with offset
         OD    16#8200_0000;  // Output Area (I/O) Code (S7)
         T     LD[AR1, P#6.0];  // ..Store byte 6/7/8/9


         LAR1;  // Load start point of cyclic data
         TAR1  #TempDword;  // Store in temp. point
         L     #TempDword;  // Load temp. point
         T     #Addr_InstanceDB;  // Store start point as DB address

         LAR1;  // Make AR1 point to calling program stack
         L     16#10;  // ANY Syntax ID
         T     LB[AR1, P#0.0];  // ..Store Byte 0
         L     16#02;  // Data Type = Byte
         T     LB[AR1, P#1.0];  // ..Store Byte 1
         L     62;  // Load Packed length
         T     LW[AR1, P#2.0];  // ..Store Byte 2/3
         L     #BlockInfo.DB_Number;  // used with DB use No. else "0"
         T     LW[AR1, P#4.0];  // ..Store byte 4/5
         L     #Addr_InstanceDB;  // Load Instance DB Start address
         L     16#8500_0000;
         -D;
         L     16#8400_0000;
         +D;
         T     LD[AR1, P#6.0];  // ..Store byte 6/7/8/9
END_REGION

REGION Network 8: Output Data to Stat area
   IF #Aoff THEN #BLOCK_RET_VAL := BLKMOV(SRCBLK := #IO_Pointer, DSTBLK => #DB_Pointer); END_IF;
END_REGION

REGION Network 9: Reset outputs in first scan
   IF NOT #TOKEN.FIRST_SCAN THEN GOTO Nres; END_IF;
END_REGION

REGION Network 10: Reset SectionOut Byte 0 and 1
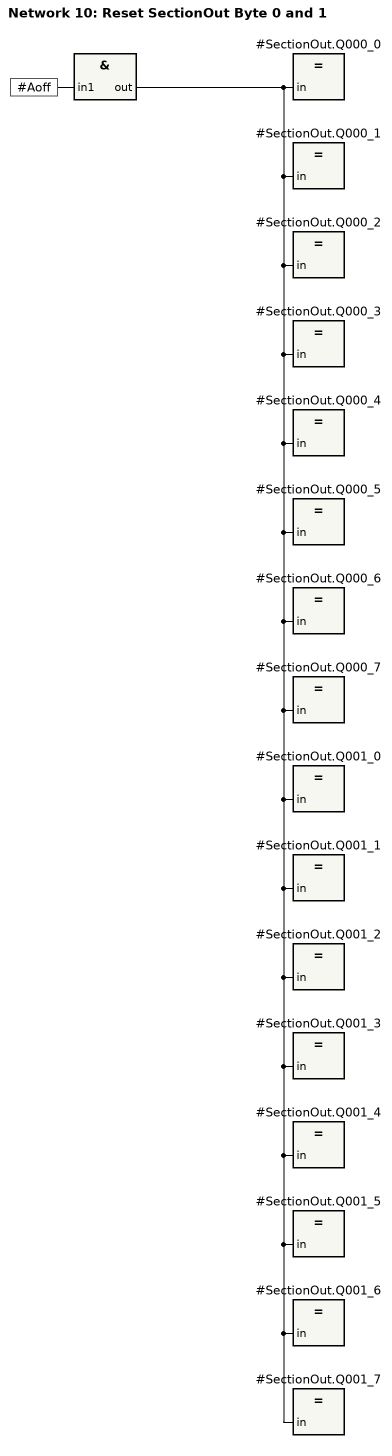
   #SectionOut.Q000_0 := #Aoff;
   #SectionOut.Q000_1 := #Aoff;
   #SectionOut.Q000_2 := #Aoff;
   #SectionOut.Q000_3 := #Aoff;
   #SectionOut.Q000_4 := #Aoff;
   #SectionOut.Q000_5 := #Aoff;
   #SectionOut.Q000_6 := #Aoff;
   #SectionOut.Q000_7 := #Aoff;
   #SectionOut.Q001_0 := #Aoff;
   #SectionOut.Q001_1 := #Aoff;
   #SectionOut.Q001_2 := #Aoff;
   #SectionOut.Q001_3 := #Aoff;
   #SectionOut.Q001_4 := #Aoff;
   #SectionOut.Q001_5 := #Aoff;
   #SectionOut.Q001_6 := #Aoff;
   #SectionOut.Q001_7 := #Aoff;
END_REGION

REGION Network 11: Reset Word 2
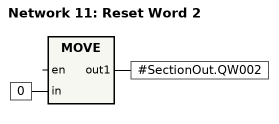
   #SectionOut.QW002 := 0;
END_REGION

REGION Network 12: Reset SectionOut Byte 4 and 5
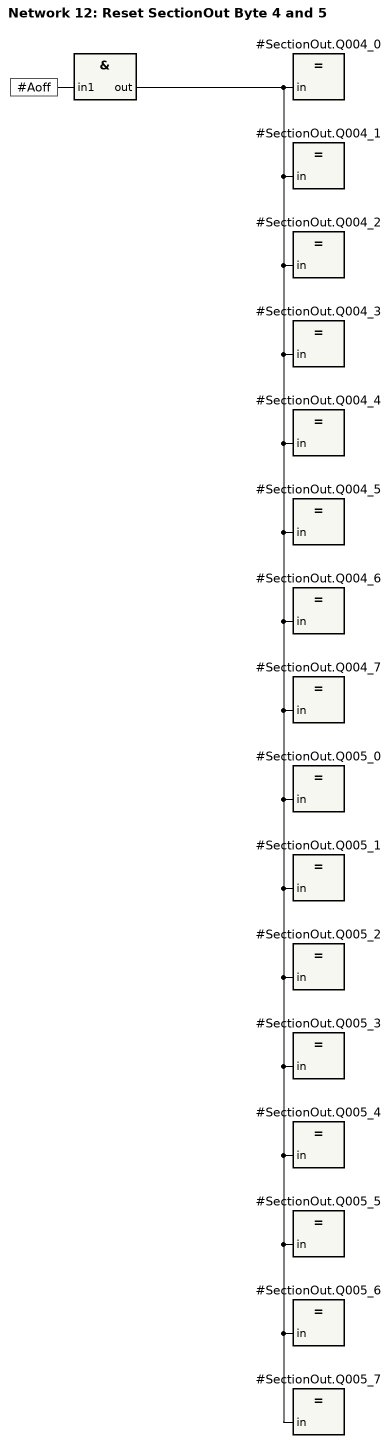
   #SectionOut.Q004_0 := #Aoff;
   #SectionOut.Q004_1 := #Aoff;
   #SectionOut.Q004_2 := #Aoff;
   #SectionOut.Q004_3 := #Aoff;
   #SectionOut.Q004_4 := #Aoff;
   #SectionOut.Q004_5 := #Aoff;
   #SectionOut.Q004_6 := #Aoff;
   #SectionOut.Q004_7 := #Aoff;
   #SectionOut.Q005_0 := #Aoff;
   #SectionOut.Q005_1 := #Aoff;
   #SectionOut.Q005_2 := #Aoff;
   #SectionOut.Q005_3 := #Aoff;
   #SectionOut.Q005_4 := #Aoff;
   #SectionOut.Q005_5 := #Aoff;
   #SectionOut.Q005_6 := #Aoff;
   #SectionOut.Q005_7 := #Aoff;
END_REGION

REGION Network 13: Reset SectionOut Byte 6 and 7
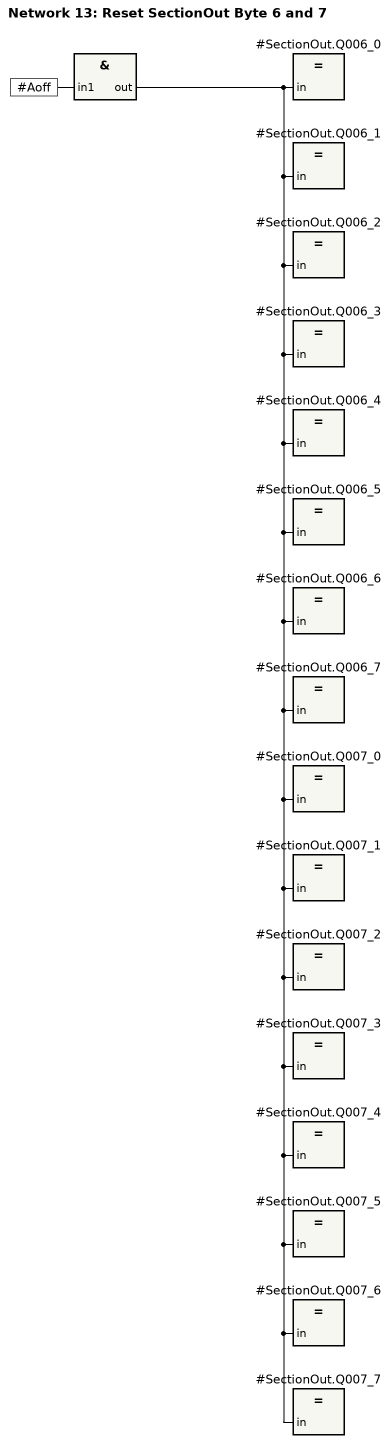
   #SectionOut.Q006_0 := #Aoff;
   #SectionOut.Q006_1 := #Aoff;
   #SectionOut.Q006_2 := #Aoff;
   #SectionOut.Q006_3 := #Aoff;
   #SectionOut.Q006_4 := #Aoff;
   #SectionOut.Q006_5 := #Aoff;
   #SectionOut.Q006_6 := #Aoff;
   #SectionOut.Q006_7 := #Aoff;
   #SectionOut.Q007_0 := #Aoff;
   #SectionOut.Q007_1 := #Aoff;
   #SectionOut.Q007_2 := #Aoff;
   #SectionOut.Q007_3 := #Aoff;
   #SectionOut.Q007_4 := #Aoff;
   #SectionOut.Q007_5 := #Aoff;
   #SectionOut.Q007_6 := #Aoff;
   #SectionOut.Q007_7 := #Aoff;
END_REGION

REGION Network 14: Reset SectionOut Byte 8 and 9
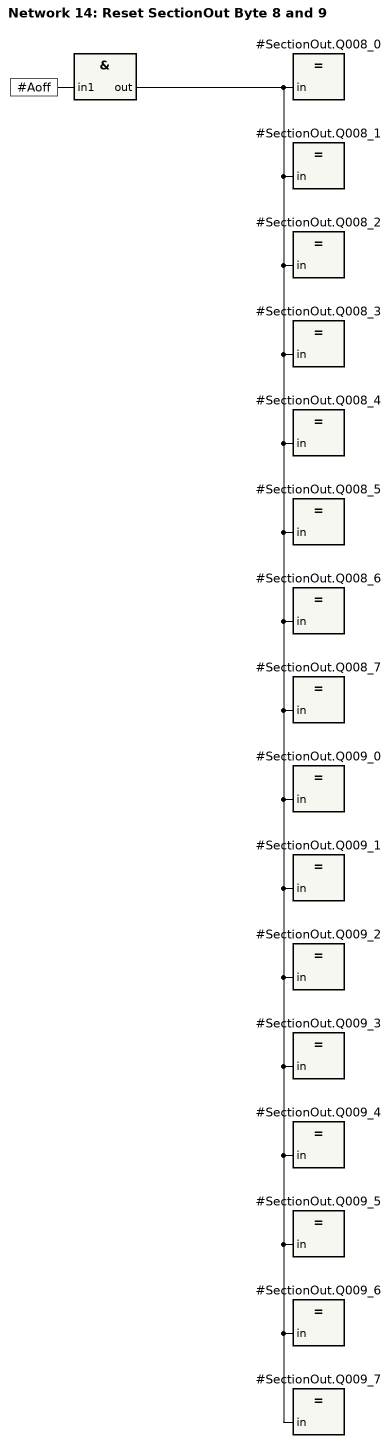
   #SectionOut.Q008_0 := #Aoff;
   #SectionOut.Q008_1 := #Aoff;
   #SectionOut.Q008_2 := #Aoff;
   #SectionOut.Q008_3 := #Aoff;
   #SectionOut.Q008_4 := #Aoff;
   #SectionOut.Q008_5 := #Aoff;
   #SectionOut.Q008_6 := #Aoff;
   #SectionOut.Q008_7 := #Aoff;
   #SectionOut.Q009_0 := #Aoff;
   #SectionOut.Q009_1 := #Aoff;
   #SectionOut.Q009_2 := #Aoff;
   #SectionOut.Q009_3 := #Aoff;
   #SectionOut.Q009_4 := #Aoff;
   #SectionOut.Q009_5 := #Aoff;
   #SectionOut.Q009_6 := #Aoff;
   #SectionOut.Q009_7 := #Aoff;
END_REGION

REGION Network 15: Reset Word 10 to 61
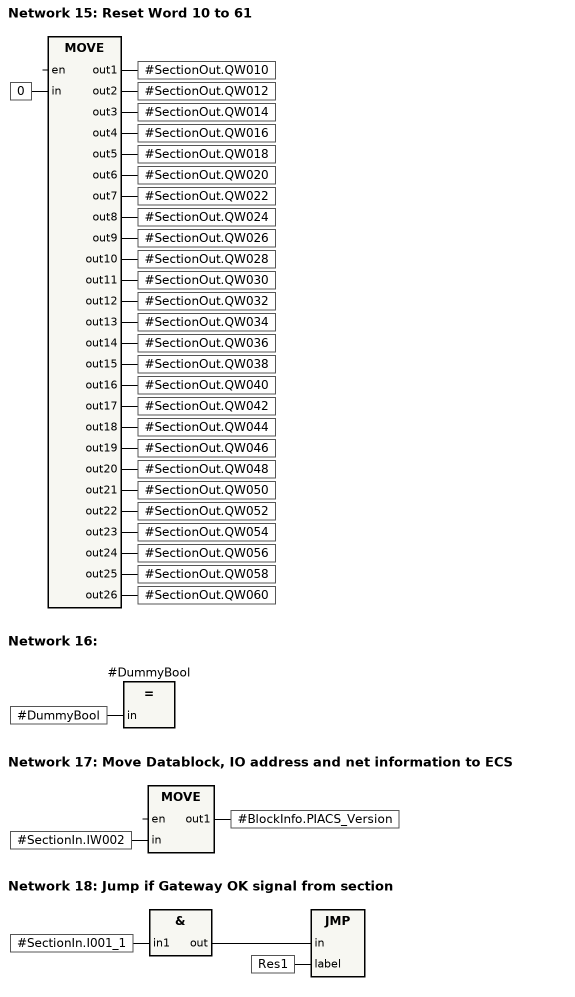
   #SectionOut.QW010 := 0;
   #SectionOut.QW012 := 0;
   #SectionOut.QW014 := 0;
   #SectionOut.QW016 := 0;
   #SectionOut.QW018 := 0;
   #SectionOut.QW020 := 0;
   #SectionOut.QW022 := 0;
   #SectionOut.QW024 := 0;
   #SectionOut.QW026 := 0;
   #SectionOut.QW028 := 0;
   #SectionOut.QW030 := 0;
   #SectionOut.QW032 := 0;
   #SectionOut.QW034 := 0;
   #SectionOut.QW036 := 0;
   #SectionOut.QW038 := 0;
   #SectionOut.QW040 := 0;
   #SectionOut.QW042 := 0;
   #SectionOut.QW044 := 0;
   #SectionOut.QW046 := 0;
   #SectionOut.QW048 := 0;
   #SectionOut.QW050 := 0;
   #SectionOut.QW052 := 0;
   #SectionOut.QW054 := 0;
   #SectionOut.QW056 := 0;
   #SectionOut.QW058 := 0;
   #SectionOut.QW060 := 0;
END_REGION

REGION Network 16
   Nres:
   #DummyBool := #DummyBool;
END_REGION

REGION Network 17: Move Datablock, IO address and net information to ECS
   #BlockInfo.PIACS_Version := #SectionIn.IW002;
END_REGION

REGION Network 18: Jump if Gateway OK signal from section
   IF #SectionIn.I001_1 THEN GOTO Res1; END_IF;
END_REGION

REGION Network 19: Reset SectionIn Byte 0 and 1
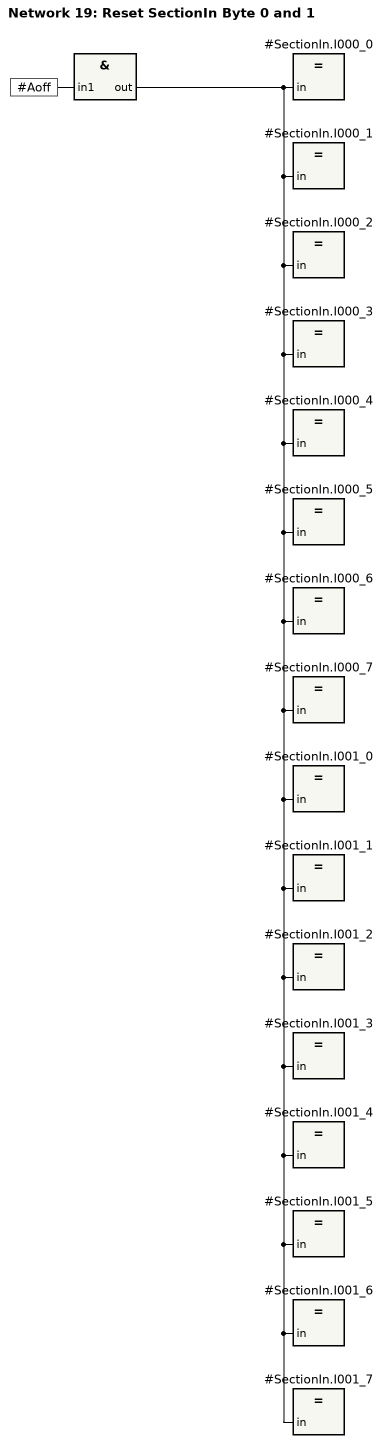
   #SectionIn.I000_0 := #Aoff;
   #SectionIn.I000_1 := #Aoff;
   #SectionIn.I000_2 := #Aoff;
   #SectionIn.I000_3 := #Aoff;
   #SectionIn.I000_4 := #Aoff;
   #SectionIn.I000_5 := #Aoff;
   #SectionIn.I000_6 := #Aoff;
   #SectionIn.I000_7 := #Aoff;
   #SectionIn.I001_0 := #Aoff;
   #SectionIn.I001_1 := #Aoff;
   #SectionIn.I001_2 := #Aoff;
   #SectionIn.I001_3 := #Aoff;
   #SectionIn.I001_4 := #Aoff;
   #SectionIn.I001_5 := #Aoff;
   #SectionIn.I001_6 := #Aoff;
   #SectionIn.I001_7 := #Aoff;
END_REGION

REGION Network 20: Reset Word 2 to 8
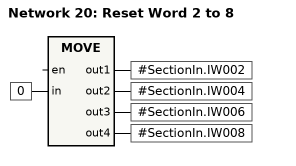
   #SectionIn.IW002 := 0;
   #SectionIn.IW004 := 0;
   #SectionIn.IW006 := 0;
   #SectionIn.IW008 := 0;
END_REGION

REGION Network 21: Reset SectionIn Byte 10 and 11
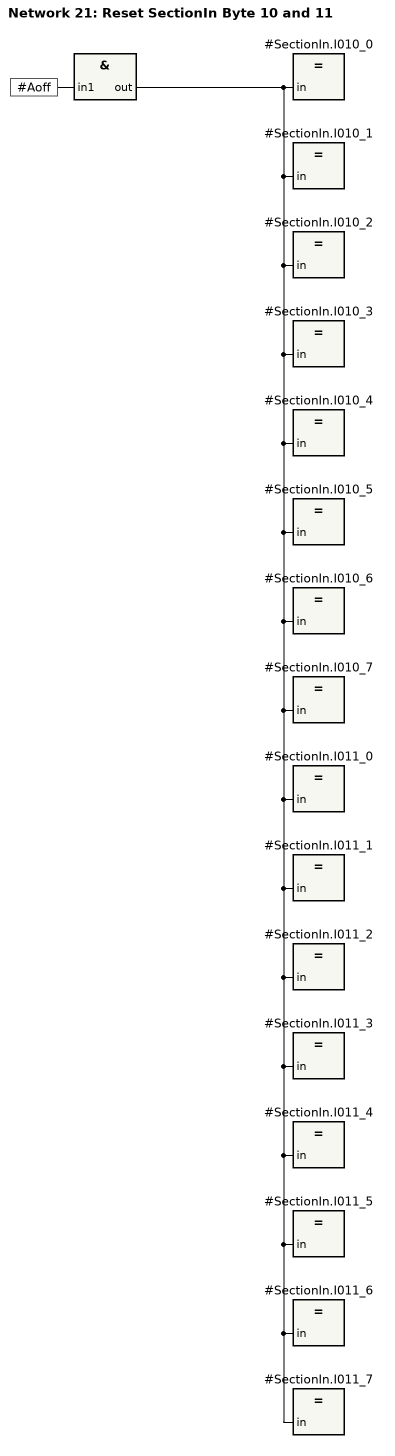
   #SectionIn.I010_0 := #Aoff;
   #SectionIn.I010_1 := #Aoff;
   #SectionIn.I010_2 := #Aoff;
   #SectionIn.I010_3 := #Aoff;
   #SectionIn.I010_4 := #Aoff;
   #SectionIn.I010_5 := #Aoff;
   #SectionIn.I010_6 := #Aoff;
   #SectionIn.I010_7 := #Aoff;
   #SectionIn.I011_0 := #Aoff;
   #SectionIn.I011_1 := #Aoff;
   #SectionIn.I011_2 := #Aoff;
   #SectionIn.I011_3 := #Aoff;
   #SectionIn.I011_4 := #Aoff;
   #SectionIn.I011_5 := #Aoff;
   #SectionIn.I011_6 := #Aoff;
   #SectionIn.I011_7 := #Aoff;
END_REGION

REGION Network 22: Reset SectionIn Byte 12 and 13
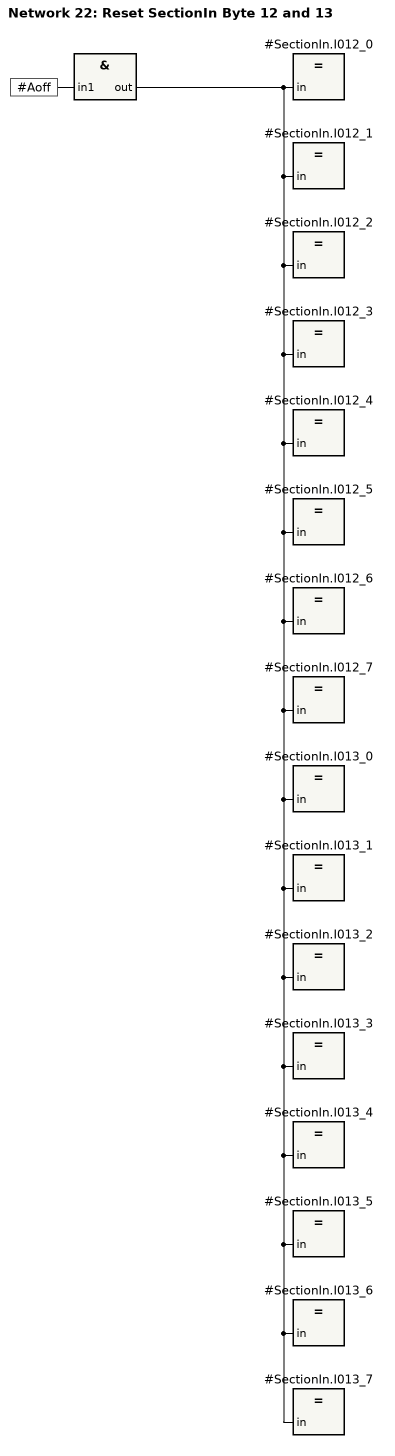
   #SectionIn.I012_0 := #Aoff;
   #SectionIn.I012_1 := #Aoff;
   #SectionIn.I012_2 := #Aoff;
   #SectionIn.I012_3 := #Aoff;
   #SectionIn.I012_4 := #Aoff;
   #SectionIn.I012_5 := #Aoff;
   #SectionIn.I012_6 := #Aoff;
   #SectionIn.I012_7 := #Aoff;
   #SectionIn.I013_0 := #Aoff;
   #SectionIn.I013_1 := #Aoff;
   #SectionIn.I013_2 := #Aoff;
   #SectionIn.I013_3 := #Aoff;
   #SectionIn.I013_4 := #Aoff;
   #SectionIn.I013_5 := #Aoff;
   #SectionIn.I013_6 := #Aoff;
   #SectionIn.I013_7 := #Aoff;
END_REGION

REGION Network 23: Reset SectionIn Byte 14 and 15
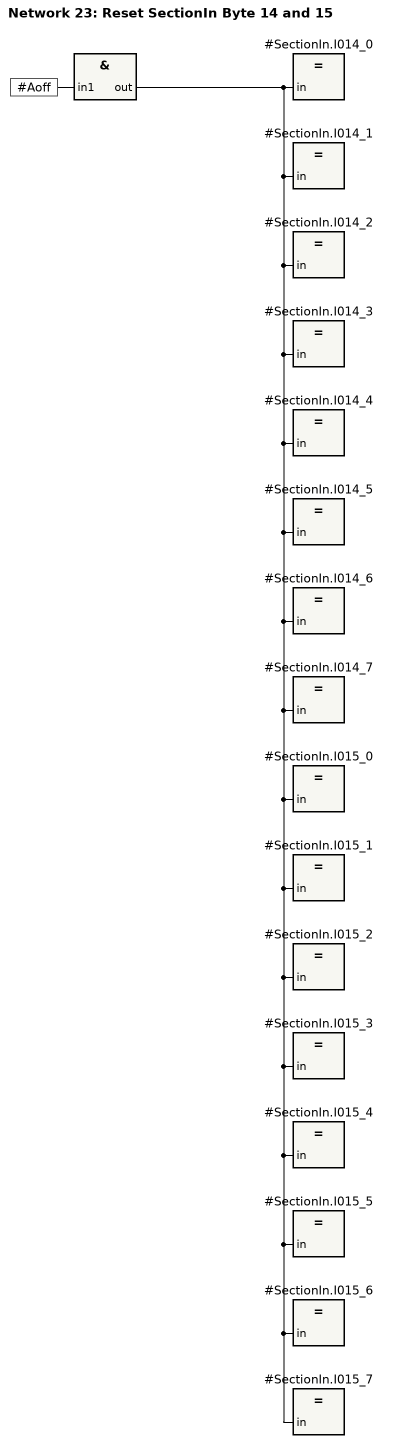
   #SectionIn.I014_0 := #Aoff;
   #SectionIn.I014_1 := #Aoff;
   #SectionIn.I014_2 := #Aoff;
   #SectionIn.I014_3 := #Aoff;
   #SectionIn.I014_4 := #Aoff;
   #SectionIn.I014_5 := #Aoff;
   #SectionIn.I014_6 := #Aoff;
   #SectionIn.I014_7 := #Aoff;
   #SectionIn.I015_0 := #Aoff;
   #SectionIn.I015_1 := #Aoff;
   #SectionIn.I015_2 := #Aoff;
   #SectionIn.I015_3 := #Aoff;
   #SectionIn.I015_4 := #Aoff;
   #SectionIn.I015_5 := #Aoff;
   #SectionIn.I015_6 := #Aoff;
   #SectionIn.I015_7 := #Aoff;
END_REGION

REGION Network 24: Reset SectionIn Byte 16 and 17
